FUNCTION_BLOCK ModbusIo
VAR_INPUT
	EN: BOOL;
	Modbus: REFERENCE TO Modbus;
	UnitID: BYTE;
	RegisterType: ModbusRegisterType;
	Register: WORD;
END_VAR
VAR_OUTPUT
	ENO: BOOL;
	Error: BOOL;
END_VAR
VAR_IN_OUT
END_VAR
VAR
	Registered: BOOL;
	ErrorCount: INT;
END_VAR
VAR PERSISTENT
END_VAR

IF EN AND __ISVALIDREF(Modbus) THEN
	IF NOT Registered THEN
		Modbus.AddIO(THIS);
		Registered := TRUE;	
	END_IF
END_IF
ENO := EN and not Error;

PROPERTY ErrorOut : BOOL
GET
ErrorOut := Error;
END_GET
SET
Error := ErrorOut;
END_SET
END_PROPERTY

METHOD GetErrorCount : INT
VAR_INPUT
END_VAR
GetErrorCount := ErrorCount;
END_METHOD

METHOD IncErrorCount : BOOL
VAR_INPUT
END_VAR
IF ErrorCount < 10 THEN
	ErrorCount := ErrorCount + 1;
END_IF
END_METHOD

METHOD ResetErrorCount : BOOL
VAR_INPUT
END_VAR
ErrorCount := 0;
END_METHOD

PROPERTY ValueBoolOut : BOOL
GET
END_GET
SET
END_SET
END_PROPERTY

PROPERTY ValueWord : WORD
GET
END_GET
SET
END_SET
END_PROPERTY

END_FUNCTION_BLOCK

(* stored: Version 1.1.0.1, ProductVersion 3.1.4024.6
   POU ModbusIo: Id {cfe7a271-9474-4996-867a-665c5c7d8c6b}, SpecialFunc None
   Property ErrorOut: Id {fba349c7-255c-4e7d-b9ff-3cd8aab40960}
   Get Get: Id {b4f378e1-a05e-4b08-b5ac-dfa8dc0c617a}
   Set Set: Id {af21a136-4472-4451-adb3-f4cea7a9b225}
   Method GetErrorCount: Id {0a7c06db-ae5c-4760-8afb-b8c2f09c3ab5}
   Method IncErrorCount: Id {ccae06b6-9936-462a-b613-d3b0d10f6e50}
   Method ResetErrorCount: Id {d0d61f1f-43b4-488b-9a90-006b7e4305c1}
   Property ValueBoolOut: Id {3afd66ea-b0f4-4521-80b0-9671f2927062}
   Get Get: Id {76813b2b-1ef4-4b99-876d-7aa6a9992400}
   Set Set: Id {678ca27f-d241-44fd-a2db-3ca3ed4711b6}
   Property ValueWord: Id {a791f941-fccb-4e94-9af3-eb1f4346b80f}
   Get Get: Id {c4f0575f-d52c-406c-8e5e-0f45d92f9f6a}
   Set Set: Id {e4efd358-cbf0-4f54-9be1-f9f72775fc2b} *)
